FUNCTION_BLOCK Camera (* Tamplate for a simple Basic Function Block Type *)
  (* Standard: 61499-2 *)
  (* Version 0.0, 2018-01-19, 4DIAC-IDE, 4DIAC-Consortium *)
  (* Version 1.0, 2016-05-26, AZ, fortiss GmbH *)
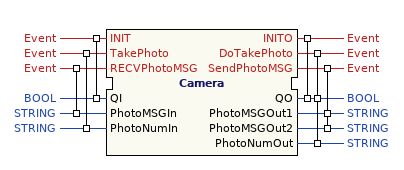
  EVENT_INPUT
    INIT WITH QI; (* Initialization Request *)
    TakePhoto WITH PhotoNumIn; (* Normal Execution Request *)
    RECVPhotoMSG WITH PhotoMSGIn;
  END_EVENT
  EVENT_OUTPUT
    INITO WITH QO; (* Initialization Confirm *)
    DoTakePhoto WITH QO, PhotoNumOut; (* Execution Confirmation *)
    SendPhotoMSG WITH PhotoMSGOut1, PhotoMSGOut2;
  END_EVENT
  VAR_INPUT
    QI : BOOL; (* Input event qualifier *)
    PhotoMSGIn : STRING;
    PhotoNumIn : STRING;
  END_VAR
  VAR_OUTPUT
    QO : BOOL; (* Output event qualifier *)
    PhotoMSGOut1 : STRING; (* pallet msg *)
    PhotoMSGOut2 : STRING; (* material msg *)
    PhotoNumOut : STRING;
  END_VAR
  VAR
    isforPallet : BOOL; (* Internal Variable *)
  END_VAR
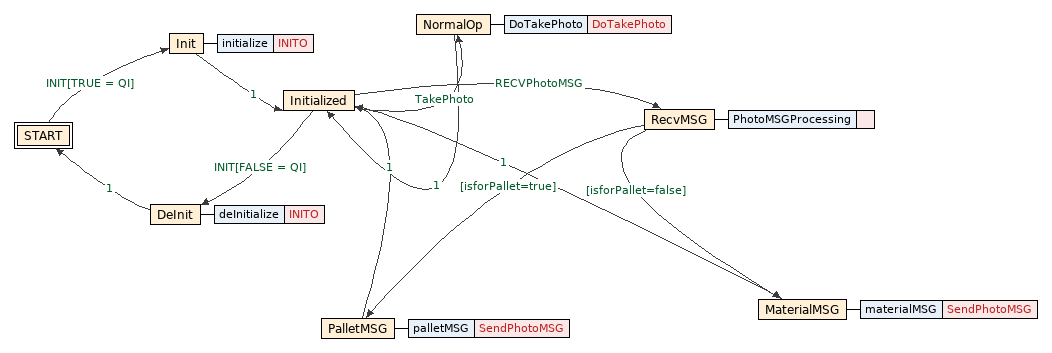
  EC_STATES
    START; (* Initial State *)
    Init : initialize -> INITO; (* Initialization *)
    NormalOp : DoTakePhoto -> DoTakePhoto; (* Normal execution *)
    Initialized;
    DeInit : deInitialize -> INITO;
    RecvMSG : PhotoMSGProcessing;
    PalletMSG : palletMSG -> SendPhotoMSG;
    MaterialMSG : materialMSG -> SendPhotoMSG;
  END_STATES
  EC_TRANSITIONS
    START TO Init := INIT[TRUE = QI];
    Init TO Initialized := 1;
    Initialized TO NormalOp := TakePhoto;
    NormalOp TO Initialized := 1;
    DeInit TO START := 1;
    Initialized TO DeInit := INIT[FALSE = QI];
    Initialized TO RecvMSG := RECVPhotoMSG;
    RecvMSG TO PalletMSG := [isforPallet=true];
    RecvMSG TO MaterialMSG := [isforPallet=false];
    PalletMSG TO Initialized := 1;
    MaterialMSG TO Initialized := 1;
  END_TRANSITIONS
  ALGORITHM initialize IN ST: (* Initialization algorithm *)
isforPallet:=true;
QO := QI;
  END_ALGORITHM
  ALGORITHM deInitialize IN ST: (* Normally executed algorithm *)
QO := FALSE;
  END_ALGORITHM
  ALGORITHM normalOperation IN ST: (* new algorithm *)
QO := QI;

IF TRUE  = QI THEN
  (*  only perform normal operation of QI is true*)

END_IF;
  END_ALGORITHM
  ALGORITHM PhotoMSGProcessing IN ST: (* new algorithm *)

  END_ALGORITHM
  ALGORITHM DoTakePhoto IN ST: (* new algorithm *)
PhotoNumOut:=PhotoNumIn;
  END_ALGORITHM
  ALGORITHM palletMSG IN ST: (* new algorithm *)
PhotoMSGOut1:=PhotoMSGIn;
  END_ALGORITHM
  ALGORITHM materialMSG IN ST: (* new algorithm *)
PhotoMSGOut2:=PhotoMSGIn;
  END_ALGORITHM
END_FUNCTION_BLOCK
